// TIA Portal project "Betriebsstundenzähler_AWL" (V16)

(* hardware
DEVICE "S71500/ET200MP station_1"  S7-1500 station
   slot 0: "Rail_0"  Rack  6ES7 590-1***0-0AA0
   slot 1: "PLC_1"  CPU 1511-1 PN  6ES7 511-1AK00-0AB0  V1.8
      slot 3: "CPU display_1"  6ES7591-1AA00-0AA0
      slot 32768: "PROFINET interface_1"  X1
         slot 32769: "Port_1"  X1 P1
         slot 32770: "Port_2"  X1 P2
   slot 2: "DI 16x24VDC BA_1"  DI 16x24VDC BA  6ES7 521-1BH10-0AA0  V1.1
*)

// ===== PLC "PLC_1"  CPU 1511-1 PN =====

VAR_GLOBAL   // PLC tag table "Default tag table"
   "Einschalttaste_Eingang" AT %I0.0 : Bool;
   "Resettaste_Eingang" AT %I0.1 : Bool;
   "Systemeinschalt_Bit" AT %M0.0 : Bool;
   "Reset_Bit" AT %M0.1 : Bool;
   "Sekunden_S" AT %MW4 : Int;
   "Sekunden_mS" AT %MD6 : DInt;
   "Minuten" AT %MW2 : Int;
   "Stunden" AT %MW10 : Int;
   "Stunden*1000" AT %MW12 : Int;
   "ONS" AT %M0.2 : Bool;
END_VAR

DATA_BLOCK "IO"   // DB1
{ S7_Optimized_Access := 'TRUE' }
VERSION : 0.1
// stored: InstanceOfName I/O
"I/O"
BEGIN
END_DATA_BLOCK

DATA_BLOCK "Steuerlogik_DB"   // DB3
{ S7_Optimized_Access := 'TRUE' }
VERSION : 0.1
// stored: InstanceOfName Steuerlogik
"Steuerlogik"
BEGIN
END_DATA_BLOCK

// folder: System blocks/Program resources

DATA_BLOCK "Timer"   // DB2
{ S7_Optimized_Access := 'TRUE' }
AUTHOR : Simatic
FAMILY : IEC
NAME : IEC_TMR
VERSION : 1.0
// stored: InstanceOfName IEC_TIMER
"IEC_TIMER"
BEGIN
END_DATA_BLOCK

DATA_BLOCK "Minuten_Zähler"   // DB4
{ S7_Optimized_Access := 'TRUE' }
AUTHOR : Simatic
FAMILY : IEC
NAME : CNTR
VERSION : 1.0
// stored: InstanceOfName IEC_COUNTER
"IEC_COUNTER"
BEGIN
END_DATA_BLOCK

DATA_BLOCK "Stunden_Zähler"   // DB5
{ S7_Optimized_Access := 'TRUE' }
AUTHOR : Simatic
FAMILY : IEC
NAME : CNTR
VERSION : 1.0
// stored: InstanceOfName IEC_COUNTER
"IEC_COUNTER"
BEGIN
END_DATA_BLOCK

DATA_BLOCK "StundenMal1000_Zähler"   // DB6
{ S7_Optimized_Access := 'TRUE' }
AUTHOR : Simatic
FAMILY : IEC
NAME : CNTR
VERSION : 1.0
// stored: InstanceOfName IEC_COUNTER
"IEC_COUNTER"
BEGIN
END_DATA_BLOCK

// folder: (top level)

FUNCTION_BLOCK "I/O"   // FB1, STL
{ S7_Optimized_Access := 'TRUE' }
VERSION : 0.1
BEGIN

REGION Network 1
         A     "Einschalttaste_Eingang";
         =     "Systemeinschalt_Bit";

         A     "Resettaste_Eingang";
         =     "Reset_Bit";
END_REGION
END_FUNCTION_BLOCK

FUNCTION_BLOCK "Steuerlogik"   // FB2, STL
{ S7_Optimized_Access := 'TRUE' }
VERSION : 0.1
   VAR
      Timer_Reset : Bool;
      TimerDone_Bit : Bool;
      Comparison : Bool;
      Minuten_Reset : Bool;
      Minuten_ZählerDone_Bit : Bool;
      ComparsionMinuten : Bool;
      Stunden_Reset : Bool;
      Stunden_ZählerDone_Bit : Bool;
      ComparisonStunden : Bool;
      StundenMal1000_Reset : Bool;
      StundenMal1000Done_Bit : Bool;
      ComparisonStundenMal1000 : Bool;
      Reset_All : Bool;
   END_VAR
BEGIN

REGION Network 1
   // Steuerlogik
   // Steuerlogik für Sekunden
         CALL  TONR, "Timer"
         ( IN := "Systemeinschalt_Bit",
           R  := #Timer_Reset,
           PT := T#60S,
           Q  := #TimerDone_Bit,
           ET :=
         );
         L     "Timer".ET;
         L     T#60S;
         <>I;
         =     #Comparison;
         A     "Systemeinschalt_Bit";
         A     #Comparison;
         L     "Timer".ET;
         T     "Sekunden_mS";
         L     "Sekunden_mS";
         L     1000;
         /D;
         T     "Sekunden_S";
         CLR;
   // Steuerlogik für Minuten
         CALL  CTU, "Minuten_Zähler"
         ( CU := #TimerDone_Bit,
           R  := #Minuten_Reset,
           PV := 60,
           Q  := #Minuten_ZählerDone_Bit,
           CV :=
         );
         L     "Minuten_Zähler".CV;
         L     60;
         <>I;
         =     #ComparsionMinuten;
         A     #ComparsionMinuten;
         L     "Minuten_Zähler".CV;
         T     "Minuten";
         CLR;
   // Steuerlogik für Stunden

         CALL  CTU ,"Stunden_Zähler"
         ( CU := #Minuten_ZählerDone_Bit,
           R  := #Stunden_Reset,
           PV := 1000,
           Q  := #Stunden_ZählerDone_Bit,
           CV :=
         );
         L     "Stunden_Zähler".CV;
         L     1000;
         <>I;
         =     #ComparisonStunden;
         A     #ComparisonStunden;
         L     "Stunden_Zähler".CV;
         T     "Stunden";
         CLR;
   //Steuerlogik für Stunden*1000

         CALL  CTU , "StundenMal1000_Zähler"
         ( CU := #Stunden_ZählerDone_Bit,
           R  := #StundenMal1000_Reset,
           PV := 1000,
           Q  := #StundenMal1000Done_Bit,
           CV :=
         );
         L     "StundenMal1000_Zähler".CV;
         L     1000;
         <>I;
         =     #ComparisonStundenMal1000;
         A     #ComparisonStundenMal1000;
         L     "StundenMal1000_Zähler".CV;
         T     "Stunden*1000";
         CLR;

   // Steuerlogik für Reset

         A     "Systemeinschalt_Bit";
         A     "Reset_Bit";
         FP    "ONS";
         =     #Reset_All;
         CLR;
         A     #TimerDone_Bit;
         O     #Reset_All;
         =     #Timer_Reset;
         CLR;
         A     #Minuten_ZählerDone_Bit;
         O     #Reset_All;
         =     #Minuten_Reset;
         CLR;
         A     #Stunden_ZählerDone_Bit;
         O     #Reset_All;
         =     #Stunden_Reset;
         A     #StundenMal1000Done_Bit;
         O     #Reset_All;
         =     #StundenMal1000_Reset;
         CLR;
END_REGION
END_FUNCTION_BLOCK

ORGANIZATION_BLOCK "Main"   // OB1, LAD, ProgramCycle
TITLE = "Main Program Sweep (Cycle)"
{ S7_Optimized_Access := 'TRUE' }
VERSION : 0.1
// PROJEKTBESCHREIBUNG:In diesem Projekt wird ein Steuerungssystem entwickelt, das die Laufzeit einer Hauptanlage erfasst. Sobald die Anlage eingeschaltet wird, beginnt der Zähler, die Betriebsdauer in Sekunden, Minuten, Hunderten und Tausenden von Stunden zu messen und in den Speicherregistern Sekunden_S, Minuten und Stunden abzulegen. Zusätzlich gibt es eine Reset-Taste, mit der der gesamte Zählerstand auf null zurückgesetzt werden kann, um eine neue Messung zu starten. Die Steuerung erfolgt über ein Einschalttaste. Solche Systeme sind essenziell, da Betriebsstunden oft als Grundlage für Wartung, Inspektion oder Garantieansprüche dienen.
// 
// TESTKRITERIEN:
// 1)Zum Starten: Führen Sie Ihr Programm in PLCSIM aus. "Sekunden_S","Minuten" und "Stunden" sollten alle auf Null stehen. Diese Werte sollten sich nicht bewegen.
// 
// 2)
// Als Nächstes erzwingen Sie den Einschalttaste_Eingang auf 1 (geschlossen). Nun sollten wir sehen, dass "Sekunden_S" akkumuliert. Es sollte immer wieder von 0 bis 59 zählen. Jedes Mal, wenn "Sekunden_S" eine Minute vollzählt, sollte "Minuten" um eins hochgehen. Irgendwann erreicht "Minuten" den Wert 59 und springt dann wieder selbst auf 0 zurück. Wenn das passiert, sollte "Stunden" um eins hochgehen. (Auch wenn wir es nicht so lange laufen lassen werden.) Nachdem "Stunden" den Wert 999 erreicht, sollte es wieder auf 0 zurückspringen und "Stunden*1000" um eins hochgehen. Und so weiter. Um zu testen, ob "Stunden" und "Stunden*1000" funktionieren, können Sie "Minuten" und "Stunden" manuell jeweils auf ihren Grenzwert setzen, um sicherzustellen, dass alles korrekt hochzählt.
// 3)
// 
// Drittens erzwingen Sie den Einschalttaste_Eingang wieder 0 (offen). Alle Ihre Akkumulatoren  sollten genau an der Stelle einfrieren, an der sie stehen.
// 
// 
// 4)Viertens erzwingen Sie den System-Run-Eingang ein letztes Mal auf 1 (geschlossen). Die Akkumulatoren sollten genau dort weiterzählen, wo sie aufgehört haben.
// 
// 
// 5)Schließlich schalten Sie Reset_Eingang EIN und dann wieder AUS. Alle Werten sollten alle auf 0 zurückgesetzt werden.
   VAR_INPUT
      Initial_Call : Bool;   // Initial call of this OB
      Remanence : Bool;   // =True, if remanent data are available
   END_VAR
BEGIN

REGION Network 1
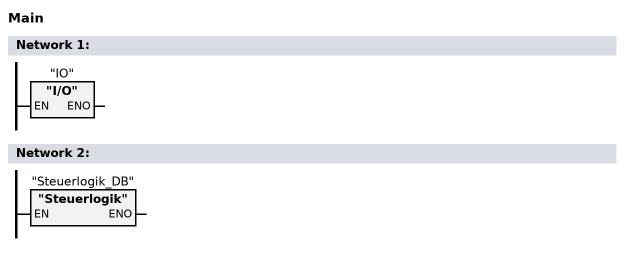
   RUNG wire#powerrail
      "IO"()
   END_RUNG
   // the same network as SCL:
   "IO"();   // "I/O"
END_REGION

REGION Network 2
   RUNG wire#powerrail
      "Steuerlogik_DB"()
   END_RUNG
   // the same network as SCL:
   "Steuerlogik_DB"();   // "Steuerlogik"
END_REGION
END_ORGANIZATION_BLOCK